FUNCTION_BLOCK EV_LinearAxis (* Typed view of LinearAxis's state channel (inputs and holder) *)
  (* Standard: 61499-2 *)
  (* Version 0.1, 2026-09-28, Project contributors, AAU Smart Production Lab *)
  PACKAGE stoppering;
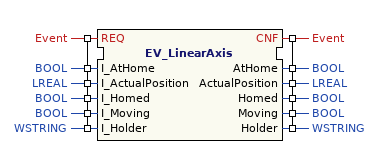
  EVENT_INPUT
    REQ WITH I_AtHome, I_ActualPosition, I_Homed, I_Moving, I_Holder;
  END_EVENT
  EVENT_OUTPUT
    CNF WITH AtHome, ActualPosition, Homed, Moving, Holder;
  END_EVENT
  VAR_INPUT
    I_AtHome : BOOL;
    I_ActualPosition : LREAL;
    I_Homed : BOOL;
    I_Moving : BOOL;
    I_Holder : WSTRING;
  END_VAR
  VAR_OUTPUT
    AtHome : BOOL;
    ActualPosition : LREAL;
    Homed : BOOL;
    Moving : BOOL;
    Holder : WSTRING;
  END_VAR
  EC_STATES
    REQ : REQ -> CNF;
  END_STATES
  ALGORITHM REQ IN ST:
AtHome := I_AtHome;
ActualPosition := I_ActualPosition;
Homed := I_Homed;
Moving := I_Moving;
Holder := I_Holder;
  END_ALGORITHM
END_FUNCTION_BLOCK
